FUNCTION_BLOCK STRIP3 (* 3-Pen Strip Chart Recorder *)
  (* Standard: 61499-1; Classification: Service Interface; ApplicationDomain: Human Interface; Function: Recorder; Type: Strip Chart *)
  (* Version 0.2, 2004-09-01, JHC, Rockwell Automation, Deleted QI, QO, MAX_SCALE, MIN_SCALE; made inputs UINT{0..100}. *)
  (* Version 0.1, 2002-05-03, JHC, Rockwell Automation, Made QI IV=true. *)
  (* Version 0.0, 2000-04-25, JHC, Rockwell Automation *)
  (* Compiler header: package fb.rt.hmi; *)
  (* Compiler Java IBM VisualAge 3.0 *)
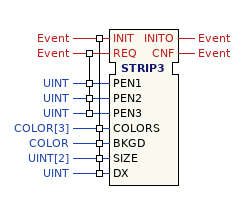
  EVENT_INPUT
    INIT WITH COLORS, BKGD, SIZE, DX;
    REQ WITH PEN1, PEN2, PEN3;
  END_EVENT
  EVENT_OUTPUT
    INITO;
    CNF;
  END_EVENT
  VAR_INPUT
    PEN1 : UINT; (* Pen 1 Position, 0-100% *)
    PEN2 : UINT; (* Pen 2 Position, 0-100% *)
    PEN3 : UINT; (* Pen 3 Position, 0-100% *)
    COLORS : ARRAY [0..2] OF COLOR := [red,yellow,green]; (* PEN1,2,3 Colors *)
    BKGD : COLOR := lightGray; (* Background Color *)
    SIZE : ARRAY [0..1] OF UINT := [200,200]; (* Width,Height *)
    DX : UINT := 10; (* x-increment size *)
  END_VAR
END_FUNCTION_BLOCK
